INTERFACE INTERNAL I_InitNode EXTENDS I_Debug;

METHOD INTERNAL Attach : Result
VAR_INPUT
	iInit		: I_InitNode;
END_VAR
END_METHOD

METHOD INTERNAL Init
VAR_OUTPUT
	iNext: I_InitNode;
END_VAR
END_METHOD

PROPERTY INTERNAL State : Result
GET
END_GET
SET
END_SET
END_PROPERTY

END_INTERFACE

(* stored: Version 1.1.0.1
   Itf I_InitNode: Id {eb6f39a4-1275-41f6-915f-4d3b3248b024}
   Method Attach: Id {3d4a1ffc-48d1-4b8d-b0fd-53f3ea042d32}
   Method Init: Id {efc19024-b584-4658-9536-3dfc6a2fb47f}
   Property State: Id {7fd1a2f9-a53e-487b-9a17-4f361344b4d4}
   Get Get: Id {dc22d531-07db-462f-ad00-3761dc7557d2}
   Set Set: Id {c58fca51-7fe1-4371-a37b-fc6ba518a207} *)
